FUNCTION_BLOCK AxDriveFB
VAR_INPUT

END_VAR
VAR_IN_OUT
	AxisController		:	AxisControl;
END_VAR
VAR_OUTPUT

END_VAR
VAR
	eCommandLatched		:	McCommand;		//Internally latched command signal, new commands cannot be issued until existing commands have completed.
											//This may need to change for sequencing
	doneLatch	:	SR;			//Used to set done signal in AxisController DUT
	bError		:	BOOL;		//Not currently implemented but may be used in future similar to bDone once more error management is implemented
	bDone		:	BOOL;		//Interal done flag which will be used for latching on an external done located in AxisController DUT
	iParam		:	INT:=1;		//index of NC parameters FBs, no 0 index on array so initialised to 1
	iIndex		:	UINT;		//index value used for limit coupling
	
	//Boolean to store EnableFw and EnableBw of MCPower FB
	FwLimitsEnabled	:	BOOL;	
	BWLimitsEnabled	:	BOOL;


//FBs as defined by PLC Open Standard
//Functions that are commented out have not been implemented yet
	//ADMIN                                                                         
	MCReset						:	MC_Reset;											
	MCPower						:	MC_Power;										
	//MCReadStatus				:	MC_ReadStatus;					//Same as Axis.ReadStatus();						
	//MCReadAxisError			:	MC_ReadAxisError;									
	MCReadParameter				:	MC_ReadParameter;									
	//MCReadBoolParameter		:	MC_ReadBoolParameter;			//not required, can be covered be McReadParameter						
	MCWriteParameter			:	MC_WriteParameter;										
	MCWriteBoolParameter		:	MC_WriteBoolParameter;								
	//MCReadDigitalInput		:	MC_ReadDigitalInput;			//NOT IMPLEMENTED		
	//MCReadDigitalOutput		:	MC_ReadDigitalOutput;			//NOT IMPLEMENTED	
	//MCWriteDigitalOutput		:	MC_WriteDigitalOutput;			//NOT IMPLEMENTED	
	//MCReadActualPosition		:	MC_ReadActualPosition;								
	//MCReadActualVelocity		:	MC_ReadActualVelocity;								
	//MCReadActualTorque		:	MC_ReadActualTorque;			//NOT IMPLEMENTED	
	//MCReadAxisInfo			:	MC_ReadAxisInfo;				//NOT IMPLEMENTED	
	//MCReadMotionState			:	MC_ReadMotionState;				//NOT IMPLEMENTED	
	MCSetPosition				:	MC_SetPosition;										
	//MCSetOverride				:	MC_SetOverride;										
	//MCTouchProbe				:	MC_TouchProbe;										
	//MCDigitalCamSwitch		:	MC_DigitalCamSwitch;			//NOT IMPLEMENTED	
	//MCAbortTrigger			:	MC_AbortTrigger;									
	//MCAbortSuperposition		:	MC_AbortSuperposition;			//HaltSuperimposed?	
	//MCCamTableSelect			:	MC_CamTableSelect;									
	
	//MCHome					:	MC_Home;											
	MCJog						:	MC_Jog;												
	//MCStop					:	MC_Stop;											
	//MCHalt					:	MC_Halt;											
	MCMoveAbsolute				:	MC_MoveAbsolute;									
	MCMoveRelative				:	MC_MoveRelative;									
	//MCMoveAdditive			:	MC_MoveAdditive;									
	//MCMoveSuperimposed		:	MC_MoveSuperimposed;								
	//MCMoveVelocity			:	MC_MoveVelocity;									
	//MCMoveContinuousAbsolute	:	MC_MoveContinuousAbsolute;						
	//MCMoveContinuousRelative	:	MC_MoveContinuousRelative;						
	//MCMoveModulo				:	MC_MoveModulo;										
	//MCTorqueControl			:	MC_TorqueControl;			//NOT IMPLEMENTED		
	//MCPositionProfile			:	MC_PositionProfile;			//NOT IMPLEMENTED		
	//MCVelocityProfile			:	MC_VelocityProfile;			//NOT IMPLEMENTED		
	//MCAccelerationProfile		:	MC_AccelerationProfile;		//NOT IMPLEMENTED		
	MCGearIn					:	MC_GearIn;											
	//MCGearInDyn				:	MC_GearInDyn;										
	MCGearInMultiMaster			:	MC_GearInMultiMaster;								
	MCGearOut					:	MC_GearOut;												                                                                                    
	//MCHaltPhasing				:	MC_HaltPhasing;										
	//MCPhasingAbsolute			:	MC_PhasingAbsolute;									
	//MCPhasingRelative			:	MC_PhasingRelative;										                                                                                                                                                 
	//MCCamIn					:	MC_CamIn;											
	//MCCamOut					:	MC_CamOut;											
	//MCCamScaling				:	MC_CamScaling;										                                                      
	//MCCamAdd					:	MC_CamAdd;											
	//MCCamExchange				:	MC_CamExchange;										
	//MCCamInV2					:	MC_CamIn_V2;		//REQUIRED FOR MULTICAMMING 	
	//MCCamRemove				:	MC_CamRemove;										
	//MCCamScalingV2			:	MC_CamScaling_V2;									

	//MOTION	
	//MCHomeRef	:	MC_StepReferencePulse;
	//MCHomeLim	:	MC_StepLimitSwitch;
	//MCHomeAbs	:	MC_StepAbsoluteSwitch;
	//homingSw	:	MC_Ref_Signal_Ref;
	//homingStruct:	MC_HomingParameter;
END_VAR

AxisController.Axis.ReadStatus();

//////////////////////////////////////////////////////////////////////
//     _   __  _____ ____    ____ _____  _  _____ _____ ____  		//
//    / \  \ \/ |_ _/ ___|  / ___|_   _|/ \|_   _| ____/ ___| 		//
//   / _ \  \  / | |\___ \  \___ \ | | / _ \ | | |  _| \___ \ 		//
//  / ___ \ /  \ | | ___) |  ___) || |/ ___ \| | | |___ ___) |		//
// /_/   \_/_/\_|___|____/  |____/ |_/_/   \_|_| |_____|____/ 		//
// 																	//
//////////////////////////////////////////////////////////////////////
                                                            
//Numerical state for axis states - may use later for buffering functions.
IF AxisController.AXIS.Status.Disabled THEN
	AxisController.iAxisState:=		100;
ELSIF AxisController.AXIS.Status.StandStill THEN
	AxisController.iAxisState:=		200;
ELSIF AxisController.AXIS.Status.Homing	THEN
	AxisController.iAxisState:= 	300;
ELSIF AxisController.AXIS.Status.DiscreteMotion	THEN
	AxisController.iAxisState:=		400;
ELSIF AxisController.AXIS.Status.SynchronizedMotion	THEN
	AxisController.iAxisState:=		500;
ELSIF AxisController.AXIS.Status.ContinuousMotion	THEN
	AxisController.iAxisState:=		600;
ELSIF AxisController.AXIS.Status.Stopping	THEN
	AxisController.iAxisState:= 	700;	
ELSIF AxisController.AXIS.Status.Error THEN
	AxisController.iAxisState:=		999;	
ELSE
	AxisController.iAxisState:=		0;
END_IF

//////////////////////////////////////////////////////////////////////////////////////////
//  _     ___ __  __ ___ _____   ______        _____ _____ ____ _   _ _____ ____  		//
// | |   |_ _|  \/  |_ _|_   _| / ___\ \      / |_ _|_   _/ ___| | | | ____/ ___| 		//
// | |    | || |\/| || |  | |   \___ \\ \ /\ / / | |  | || |   | |_| |  _| \___ \ 		//
// | |___ | || |  | || |  | |    ___) |\ V  V /  | |  | || |___|  _  | |___ ___) |		//
// |_____|___|_|  |_|___| |_|   |____/  \_/\_/  |___| |_| \____|_| |_|_____|____/		//
//																						//
//////////////////////////////////////////////////////////////////////////////////////////
//Set EnableFW and EnableBW flags based on axis limit states to begin
FwLimitsEnabled :=Limits.FwLimit[AxisController.Axis.NcToPlc.AxisId];
BwLimitsEnabled :=Limits.BwLimit[AxisController.Axis.NcToPlc.AxisId];

//Allow Master axes to listen to slave axes
//Look through array structure that manages forward and backward coupling for axis, if a slave is present check whether it is
//a FW limit or BW limit that matters and compare this against the hardware status.
//This check used to use the AxisID value from the NC however this had issues as incorrectly set NC IDs would break
//A GVL is now used to check what axis we are currently running
FOR iIndex:=1 TO GVL.axisNumMax BY 1 DO
	IF Limits.FwLimitsCoupling[GVL.iAxis][iIndex]= limitCoupling.FwSw AND NOT Limits.FwLimit[iIndex] THEN
		FwLimitsEnabled:=FALSE;
	END_IF
	IF Limits.FwLimitsCoupling[GVL.iAxis][iIndex]= limitCoupling.BwSw AND NOT Limits.BwLimit[iIndex] THEN
		FwLimitsEnabled:=FALSE;
	END_IF
	IF Limits.BwLimitsCoupling[GVL.iAxis][iIndex]= limitCoupling.BwSw AND NOT Limits.BwLimit[iIndex] THEN
		BwLimitsEnabled:=FALSE;
	END_IF
	IF Limits.BwLimitsCoupling[GVL.iAxis][iIndex]= limitCoupling.FwSw AND NOT Limits.FwLimit[iIndex] THEN
		BwLimitsEnabled:=FALSE;
	END_IF
END_FOR

//////////////////////////////////////////////////////////
//  ____   _____        _______ ____    _   _ ____  	//
// |  _ \ / _ \ \      / | ____|  _ \  | | | |  _ \ 	//
// | |_) | | | \ \ /\ / /|  _| | |_) | | | | | |_) |	//
// |  __/| |_| |\ V  V / | |___|  _ <  | |_| |  __/ 	//
// |_|    \___/  \_/\_/  |_____|_| \_\  \___/|_|   		//
//														//
/////////////////////////////////////////////////////////// 
                                               
MCPower(
	Axis:=AxisController.Axis,
	Enable:=AxisController.bEnable,
	Enable_Positive:=FwLimitsEnabled,
	Enable_Negative:=BwLimitsEnabled,
	Override:=AxisController.fOverride,
	Status=>,
	Busy=>, 
	Active=>AxisController.bAxisReady,	//Maybe want a bPowered or bEnabled flag instead?
	Error=>,
	ErrorID=>
);


//////////////////////////////////////////////////////////////////////////////////////////////////////////
//  ____  _____    _    ____    ____   _    ____     _    __  __ _____ _____ _____ ____  ____  			//
// |  _ \| ____|  / \  |  _ \  |  _ \ / \  |  _ \   / \  |  \/  | ____|_   _| ____|  _ \/ ___| 			//
// | |_) |  _|   / _ \ | | | | | |_) / _ \ | |_) | / _ \ | |\/| |  _|   | | |  _| | |_) \___ \ 			//
// |  _ <| |___ / ___ \| |_| | |  __/ ___ \|  _ < / ___ \| |  | | |___  | | | |___|  _ < ___) |			//
// |_| \_|_____/_/   \_|____/  |_| /_/   \_|_| \_/_/   \_|_|  |_|_____| |_| |_____|_| \_|____/ 			//
//                                                                                           			//
//////////////////////////////////////////////////////////////////////////////////////////////////////////
//Read in motion parameters: cycle through the 17 available
MCReadParameter(Axis:=AxisController.AXIS,ParameterNumber:=iParam);
IF MCReadParameter.Valid THEN
	MCReadParameter.Enable:=FALSE;
	AxisController.fParametersOut[iParam]:=MCReadParameter.Value;
	iParam:= iParam+1;
	IF iParam>17 THEN
		iParam:=1;
	END_IF
ELSE
	MCReadParameter.Enable:=TRUE;
END_IF

//To save on using a separate bool parameter read just converting the REALs to BOOLS and storing in flags
IF AxisController.fParametersOut[RWParameter.EnableLimitPos]=1 THEN
	AxisController.bSoftLimPosEn:=TRUE;
ELSE
	AxisController.bSoftLimPosEn:=FALSE;
END_IF

IF AxisController.fParametersOut[RWParameter.EnableLimitNeg]=1 THEN
	AxisController.bSoftLimNegEn:=TRUE;
ELSE
	AxisController.bSoftLimNegEn:=FALSE;
END_IF

IF AxisController.fParametersOut[RWParameter.EnablePosLagMonitoring]=1 THEN
	AxisController.bPosLagEn:=TRUE;
ELSE
	AxisController.bPosLagEn:=FALSE;
END_IF

//////////////////////////////////////////////////////////////////////////////////////////////////////////
//  __  __  ____   _____ _   _ _   _  ____ _____ ___ ___  _   _    ____    _    _     _     ____  		//
// |  \/  |/ ___| |  ___| | | | \ | |/ ___|_   _|_ _/ _ \| \ | |  / ___|  / \  | |   | |   / ___| 		//
// | |\/| | |     | |_  | | | |  \| | |     | |  | | | | |  \| | | |     / _ \ | |   | |   \___ \ 		//
// | |  | | |___  |  _| | |_| | |\  | |___  | |  | | |_| | |\  | | |___ / ___ \| |___| |___ ___) |		//
// |_|  |_|\____| |_|    \___/|_| \_|\____| |_| |___\___/|_| \_|  \____/_/   \_|_____|_____|____/ 		//
//                                         																//                                                      
//////////////////////////////////////////////////////////////////////////////////////////////////////////
//Call MC Function Blocks and clear execute signals
//Function blocks will hold done and error signals for 1 cycle with no execute held
MCReadParameter(Axis:=AxisController.Axis);	//Reading in motion parameters, using one functionblock for all params means need to disable
MCReset(Axis:=AxisController.Axis);
MCReset.Execute:=FALSE;
MCWriteParameter(Axis:=AxisController.Axis);
MCWriteParameter.Execute:=FALSE;
MCWriteBoolParameter(Axis:=AxisController.Axis);
MCWriteBoolParameter.Execute:=FALSE;
MCSetPosition(Axis:=AxisController.Axis);
MCSetPosition.Execute:=FALSE;
MCMoveAbsolute(Axis:=AxisController.Axis);
MCMoveAbsolute.Execute:=FALSE;
MCMoveRelative(Axis:=AxisController.Axis);
MCMoveRelative.Execute:=FALSE;
MCGearIn(Slave:=AxisController.Axis, Master:=AxisController.masterAxis);
MCGearIn.Execute:=FALSE;
MCGearInMultiMaster(Master1:=AxisController.masterAxis1,Master2:=AxisController.masterAxis2,Master3:=AxisController.masterAxis3,Master4:=AxisController.masterAxis4,Slave:=AxisController.Axis);
MCGearInMultiMaster.Enable:=FALSE;	//NOT EXECUTE AS FB ALLOWS CONTINUAL UPDATING OF RATIOS WHILST ENABLED, testing move here
MCGearOut(Slave:=AxisController.Axis);
MCGearOut.Execute:=FALSE;
MCJog(Axis:=AxisController.Axis);
MCJog.JogBackwards:=FALSE;
MCJog.JogForward:=FALSE;

//If we're not doing anything or have just done something we no longer latch on the given command
IF NOT AxisController.AXIS.Status.HasJob OR AxisController.bDone THEN
	eCommandLatched:=AxisController.eCommand;
END_IF



//////////////////////////////////////////////////////////////////////////////////////////////////////////////////////////////////////////////
//   ____ ___  __  __ __  __    _    _   _ ____     ____    _    ____  _____   ____ _____  _  _____ _____ __  __ _____ _   _ _____ ____ 	// 
//  / ___/ _ \|  \/  |  \/  |  / \  | \ | |  _ \   / ___|  / \  / ___|| ____| / ___|_   _|/ \|_   _| ____|  \/  | ____| \ | |_   _/ ___| 	//
// | |  | | | | |\/| | |\/| | / _ \ |  \| | | | | | |     / _ \ \___ \|  _|   \___ \ | | / _ \ | | |  _| | |\/| |  _| |  \| | | | \___ \ 	//
// | |__| |_| | |  | | |  | |/ ___ \| |\  | |_| | | |___ / ___ \ ___) | |___   ___) || |/ ___ \| | | |___| |  | | |___| |\  | | |  ___) |	//
//  \____\___/|_|  |_|_|  |_/_/   \_|_| \_|____/   \____/_/   \_|____/|_____| |____/ |_/_/   \_|_| |_____|_|  |_|_____|_| \_| |_| |____/	//
//																																			//
//////////////////////////////////////////////////////////////////////////////////////////////////////////////////////////////////////////////
CASE eCommandLatched OF
	
	MCCommand.Idle:
		AxisController.bBusy	:=FALSE;
		AxisController.bExecute	:=FALSE;
///////////////////////////////////////////////////////////////////////////////////////////////////////////////////////////////	
	MCCommand.Reset:
		AxisController.bError	:=FALSE;
		MCReset.Execute:=AxisController.bReset;
		bDone:=McReset.Done;
		AxisController.bBusy:=MCReset.Busy;
		IF MCReset.Error THEN
			AxisController.bError:=TRUE;
			AxisController.iErrorID:=MCReset.ErrorID;	
		END_IF
		
		//Clear command and erase reset flag.
		IF NOT MCReset.Busy THEN
			eCommandLatched:=MCCommand.Idle;
			AxisController.bReset:=FALSE;
		END_IF
///////////////////////////////////////////////////////////////////////////////////////////////////////////////////////////////
	MCCommand.WriteParameter:		
		MCWriteParameter.Execute:=AxisController.bExecute;
		MCWriteParameter.ParameterNumber:=AxisController.iParameterIndex;
		MCWriteParameter.Value:=AxisController.fParameterValue;
		bDone:=MCWriteParameter.Done;
		AxisController.bBusy:= MCWriteParameter.Busy;
		IF MCWriteParameter.Error THEN
			AxisController.bError:=TRUE;
			AxisController.iErrorID:=MCWriteParameter.ErrorID;	
		END_IF
		
		IF NOT MCWriteParameter.Busy THEN
			eCommandLatched:=MCCommand.Idle;
		END_IF			
///////////////////////////////////////////////////////////////////////////////////////////////////////////////////////////////
	MCCommand.WriteBoolParameter:	
		MCWriteBoolParameter.Execute:=AxisController.bExecute;
		MCWriteBoolParameter.ParameterNumber:=AxisController.iParameterIndex;
		MCWriteBoolParameter.Value:=AxisController.bInput;
		bDone:=MCWriteBoolParameter.Done;
		AxisController.bBusy:=MCWriteBoolParameter.Busy;
		
		IF MCWriteBoolParameter.Error THEN
			AxisController.bError:= TRUE;
			AxisController.iErrorID:=MCWriteBoolParameter.ErrorID;
		END_IF
				
		IF NOT MCWriteBoolParameter.Busy THEN
			eCommandLatched:=MCCommand.Idle;
		END_IF	
///////////////////////////////////////////////////////////////////////////////////////////////////////////////////////////////
	MCCommand.SetPosition:	
		MCSetPosition.Execute:=AxisController.bExecute;
		MCSetPosition.Position:=AxisController.fPosition;
		AxisController.bBusy:=MCSetPosition.Busy;
		bDone:=MCSetPosition.Done;
		IF MCSetPosition.Error THEN
			AxisController.bError:=TRUE;
			AxisController.iErrorID:= MCSetPosition.ErrorID;
		END_IF
		IF NOT MCSetPosition.Busy THEN
			eCommandLatched:=MCCommand.Idle;
		END_IF
///////////////////////////////////////////////////////////////////////////////////////////////////////////////////////////////
	MCCommand.MoveAbsolute:	
		MCMoveAbsolute.Execute:=AxisController.bExecute;
		MCMoveAbsolute.Position:=AxisController.fPosition;
		MCMoveAbsolute.Velocity:=AxisController.fVelocity;
		MCMoveAbsolute.Acceleration:=AxisController.fAcceleration;
		MCMoveAbsolute.Deceleration:=AxisController.fDeceleration;
		MCMoveAbsolute.Jerk:=0;
		MCMoveAbsolute.BufferMode:=MC_BufferMode.MC_Buffered;
		
		bDone:=MCMoveAbsolute.Done;
		AxisController.bBusy:=MCMoveAbsolute.Busy;
		
		IF MCMoveAbsolute.Error THEN
			AxisController.bError:=TRUE;
			AxisController.iErrorID:=MCMoveAbsolute.ErrorID;
		END_IF
		IF NOT MCMoveAbsolute.Busy THEN
			eCommandLatched:=MCCommand.Idle;
		END_IF
///////////////////////////////////////////////////////////////////////////////////////////////////////////////////////////////
	MCCommand.MoveRelative:		//MOVE RELATIVE
		MCMoveRelative.Execute:=AxisController.bExecute;
		MCMoveRelative.Distance:=AxisController.fDistance;
		MCMoveRelative.Velocity:=AxisController.fVelocity;
		MCMoveRelative.Acceleration:=AxisController.fAcceleration;
		MCMoveRelative.Deceleration:=AxisController.fDeceleration;
		MCMoveRelative.Jerk:=0;
		MCMoveRelative.BufferMode:=MC_BufferMode.MC_Buffered;
		bDone:=MCMoveRelative.Done;
		AxisController.bBusy:=MCMoveRelative.Busy;
		IF MCMoveRelative.Error THEN
			AxisController.bError:=TRUE;
			AxisController.iErrorID:=MCMoveRelative.ErrorID;
		END_IF
		IF NOT MCMoveRelative.Busy THEN
			eCommandLatched:=MCCommand.Idle;
		END_IF		
///////////////////////////////////////////////////////////////////////////////////////////////////////////////////////////////
	MCCommand.GearIn:
	
		//Dependent on +ve or -ve gear ratio determines whether to link Fw to Fw and Bw to Bw or Fw to Bw and Bw to Fw
		IF AxisController.fGearRatioNum>0 THEN
			Limits.FwLimitsCoupling[AxisController.masterAxis.NcToPlc.AxisId][AxisController.Axis.NcToPlc.AxisId]:=limitCoupling.FwSw;
			Limits.BwLimitsCoupling[AxisController.masterAxis.NcToPlc.AxisId][AxisController.Axis.NcToPlc.AxisId]:=limitCoupling.BwSw;
		END_IF
		IF AxisController.fGearRatioNum<0 THEN
			Limits.FwLimitsCoupling[AxisController.masterAxis.NcToPlc.AxisId][AxisController.Axis.NcToPlc.AxisId]:=limitCoupling.BwSw;
			Limits.BwLimitsCoupling[AxisController.masterAxis.NcToPlc.AxisId][AxisController.Axis.NcToPlc.AxisId]:=LimitCoupling.FwSw;
		END_IF
		
		MCGearIn.Execute:=AxisController.bExecute;
		MCGearIn.RatioNumerator:=AxisController.fGearRatioNum;
		MCGearIn.RatioDenominator:=AxisController.iGearRatioDen;
		AxisController.bBusy:=MCGearIn.Busy;
		IF MCGearIn.Error THEN
			AxisController.bError:=TRUE;
			AxisController.iErrorID:=MCGearIn.ErrorID;
		END_IF
		bDone:=McGearIn.InGear;
		IF NOT MCGearIn.Busy THEN
			eCommandLatched:=MCCommand.Idle;
		END_IF
///////////////////////////////////////////////////////////////////////////////////////////////////////////////////////////////
	MCCommand.GearInMultiMaster:
		IF AxisController.fGearRatio1>0 THEN
			Limits.FwLimitsCoupling[AxisController.masterAxis1.NcToPlc.AxisId][AxisController.Axis.NcToPlc.AxisId]:=limitCoupling.FwSw;
			Limits.BwLimitsCoupling[AxisController.masterAxis1.NcToPlc.AxisId][AxisController.Axis.NcToPlc.AxisId]:=limitCoupling.BwSw;
		END_IF
		IF AxisController.fGearRatio1<0 THEN
			Limits.FwLimitsCoupling[AxisController.masterAxis1.NcToPlc.AxisId][AxisController.Axis.NcToPlc.AxisId]:=limitCoupling.BwSw;
			Limits.BwLimitsCoupling[AxisController.masterAxis1.NcToPlc.AxisId][AxisController.Axis.NcToPlc.AxisId]:=LimitCoupling.FwSw;
		END_IF
		IF AxisController.fGearRatio2>0 THEN
			Limits.FwLimitsCoupling[AxisController.masterAxis2.NcToPlc.AxisId][AxisController.Axis.NcToPlc.AxisId]:=limitCoupling.FwSw;
			Limits.BwLimitsCoupling[AxisController.masterAxis2.NcToPlc.AxisId][AxisController.Axis.NcToPlc.AxisId]:=limitCoupling.BwSw;
		END_IF
		IF AxisController.fGearRatio2<0 THEN
			Limits.FwLimitsCoupling[AxisController.masterAxis2.NcToPlc.AxisId][AxisController.Axis.NcToPlc.AxisId]:=limitCoupling.BwSw;
			Limits.BwLimitsCoupling[AxisController.masterAxis2.NcToPlc.AxisId][AxisController.Axis.NcToPlc.AxisId]:=LimitCoupling.FwSw;
		END_IF
		IF AxisController.fGearRatio3>0 THEN
			Limits.FwLimitsCoupling[AxisController.masterAxis3.NcToPlc.AxisId][AxisController.Axis.NcToPlc.AxisId]:=limitCoupling.FwSw;
			Limits.BwLimitsCoupling[AxisController.masterAxis3.NcToPlc.AxisId][AxisController.Axis.NcToPlc.AxisId]:=limitCoupling.BwSw;
		END_IF
		IF AxisController.fGearRatio3<0 THEN
			Limits.FwLimitsCoupling[AxisController.masterAxis3.NcToPlc.AxisId][AxisController.Axis.NcToPlc.AxisId]:=limitCoupling.BwSw;
			Limits.BwLimitsCoupling[AxisController.masterAxis3.NcToPlc.AxisId][AxisController.Axis.NcToPlc.AxisId]:=LimitCoupling.FwSw;
		END_IF
		IF AxisController.fGearRatio4>0 THEN
			Limits.FwLimitsCoupling[AxisController.masterAxis4.NcToPlc.AxisId][AxisController.Axis.NcToPlc.AxisId]:=limitCoupling.FwSw;
			Limits.BwLimitsCoupling[AxisController.masterAxis4.NcToPlc.AxisId][AxisController.Axis.NcToPlc.AxisId]:=limitCoupling.BwSw;
		END_IF
		IF AxisController.fGearRatio4<0 THEN
			Limits.FwLimitsCoupling[AxisController.masterAxis4.NcToPlc.AxisId][AxisController.Axis.NcToPlc.AxisId]:=limitCoupling.BwSw;
			Limits.BwLimitsCoupling[AxisController.masterAxis4.NcToPlc.AxisId][AxisController.Axis.NcToPlc.AxisId]:=LimitCoupling.FwSw;
		END_IF
		
		//issue with this MC block (other than everything...) is that it doesn't conform to the standard and use an execute signal. The execute
		//signal in any other block determines that when it is high one of either error,done,busy must be on. That is not the case with this block
		//what happens is it triggers, doesn't register a busy and so immediately clears as done.
		
		MCGearInMultiMaster.Enable:=AxisController.bExecute;
		MCGearInMultiMaster.GearRatio1:=AxisController.fGearRatio1;
		MCGearInMultiMaster.GearRatio2:=AxisController.fGearRatio2;
		MCGearInMultiMaster.GearRatio3:=AxisController.fGearRatio3;
		MCGearInMultiMaster.GearRatio4:=AxisController.fGearRatio4;
		
		AxisController.bBusy:=MCGearInMultiMaster.Busy;
		IF MCGearInMultiMaster.Enable THEN
			AxisController.bBusy:=TRUE;	//busy does not go immediately high when enable high 
			bDone:=FALSE;
		END_IF

		bDone:=MCGearInMultiMaster.InGear;	// This does not work, the InGear seems to trigger before they are in gear, "active" flag does not work either.
		IF MCGearInMultiMaster.Error THEN
			AxisController.bError:=TRUE;
			AxisController.iErrorID:=MCGearInMultiMaster.ErrorID;
		END_IF
		IF NOT MCGearInMultiMaster.Busy THEN
			eCommandLatched:=MCCommand.Idle;
		END_IF
///////////////////////////////////////////////////////////////////////////////////////////////////////////////////////////////
	MCCommand.GearOut:
		//Clear limit link of this slave to master. Cycle through all master arrays clearing link
		FOR iIndex:=1 TO GVL.axisNumMax BY 1 DO
			Limits.FwLimitsCoupling[iIndex][AxisController.Axis.NcToPlc.AxisId]:=LimitCoupling.None;
			Limits.BwLimitsCoupling[iIndex][AxisController.Axis.NcToPlc.AxisId]:=LimitCoupling.None;
		END_FOR
		
		MCGearOut.Execute:=AxisController.bExecute;
		AxisController.bBusy:=MCGearOut.Busy;
		bDone:=MCGearOut.Done;
		IF MCGearOut.Error THEN
			AxisController.bError:=TRUE;
			AxisController.iErrorID:=MCGearOut.ErrorID;
		END_IF
		IF NOT MCGearOut.Busy THEN
			eCommandLatched:=MCCommand.Idle;
		END_IF
	///////////////////////////////////////////////////////////////////////////////////////////////////////////////////////////////			
	MCCommand.Jog:
		MCJog.JogForward:=AxisController.bJogForward;
		MCJog.JogBackwards:=AxisController.bJogBackward;
		bDone:=MCJog.Done;
		IF MCJog.Error THEN
			AxisController.bError:=TRUE;
			AxisController.iErrorID:=MCJog.ErrorID;
		END_IF
		IF NOT MCJog.Busy THEN
			eCommandLatched:=MCCommand.Idle;
		END_IF

END_CASE

////////////////////////////////////////// 
//  _____ _        _    ____ ____  		//
// |  ___| |      / \  / ___/ ___| 		//
// | |_  | |     / _ \| |  _\___ \ 		//
// |  _| | |___ / ___ | |_| |___) |		//
// |_|   |_____/_/   \_\____|____/ 		//
//                                		//
//////////////////////////////////////////
AxisController.bMoving:=AxisController.Axis.Status.Moving;

//Logic to latch on the done signal. As per the standard, unless the execute line is held high, there will be no done 
//output, so this latches that signal the one cycle it is on.
//doneLatch(SET1:=bDone,RESET:=AxisController.bBUSY OR AxisController.bERROR);
//AxisController.latchDONE:=doneLatch.Q1;
//
//errorLatch(SET1:=AxisController.bERROR, RESET:=AxisController.bBUSY OR bDone);
//AxisController.latchERROR:=errorLatch.Q1;

			
AxisController.bExecute:=FALSE;



doneLatch(SET1:=bDone,RESET:=(AxisController.bBusy OR AxisController.bError));
AxisController.bDone:=doneLatch.Q1;

END_FUNCTION_BLOCK

(* stored: Version 1.1.0.1, ProductVersion 3.1.4020.12
   POU AxDriveFB: Id {aef7aef0-3971-449b-83a3-6f8c4c2f7d04}, SpecialFunc None *)
